FUNCTION F_OR_REF_EX : BOOL
VAR_IN_OUT
	bValueRoot		: BOOL;	
END_VAR
VAR_INPUT
	bValueCombine	: BOOL;
	bInitialize		: BOOL;
END_VAR

IF bInitialize THEN
	bValueRoot := FALSE;
END_IF

F_OR_REF(bValueRoot, bValueCombine);

END_FUNCTION

(* stored: Version 1.1.0.1, ProductVersion 3.1.4024.11
   POU F_OR_REF_EX: Id {caae6390-40ff-47bf-87c8-b8e466592888}, SpecialFunc None *)
